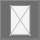
VISUALIZATION _VISU_ButtonFrameSel  // 40x40
VAR_IN_OUT
  mCfg : ST_ButtonFrameSel_Def;
END_VAR
    RoundedRectangle (0,0 40x40), tooltip "%s", colour toggle: mCfg.pFrameSelect^ = mCfg.nFrameIdx
        p4168582468: mCfg.sVisuName
        OnMouseClick: execute { mCfg.pFrameSelect^ := mCfg.nFrameIdx; }
    Image (10,5 20x30), tooltip "%s"
        p84334746: mCfg.sImgId
        p4168582468: mCfg.sVisuName
        OnMouseClick: execute { mCfg.pFrameSelect^ := mCfg.nFrameIdx; }
END_VISUALIZATION

(* stored: Version 1.1.0.1, ProductVersion 3.1.4024.11
   Visu _VISU_ButtonFrameSel: Id {64768199-8b5a-48c8-94e5-61b61ed51969} *)
